FUNCTION_BLOCK FB_PcShutdownController
VAR
//---FB_Initで受け取り---
	_pPersistentDataManager		:POINTER TO FB_PersistentDataManager;		//パーシステントデータ書き込み
	_PcAmsNetId					:AMSNETID;									//PC AMS Net ID	

//---内部使用FB---
	fbPlcStop					:PLC_Stop		:=(Stop:=FALSE);			//PLCストップ
	fbNtShutdown				:NT_Shutdown	:=(START:=FALSE);			//PCシャットダウン
	fbNtReboot					:NT_Reboot		:=(START:=FALSE);			//PCリブート

	fbRebootTon					:TON			:=(PT:=T#2S);
	fbShutdownTon				:TON			:=(PT:=T#2S);
	
//---内部変数---
	iStep						:INT			:=0;						//シャットダウン、リブート制御step
	_bError						:BOOL;
	_bReboot					:BOOL;
	_bShutdown					:BOOL;
END_VAR

PROPERTY bError : BOOL
GET
bError:=_bError;
END_GET
END_PROPERTY

METHOD Execute
//---パーシステントデータ保存FBのポインターチェック---
	IF _pPersistentDataManager=0 THEN
		_bError:=TRUE;
		iStep:=0;
		RETURN;
		
	END_IF	



//---タイマーFB呼び出し---
	fbRebootTon(IN:=_bReboot AND NOT _bShutdown AND NOT _bError );
	fbShutdownTon(IN:=_bShutdown AND NOT _bReboot AND NOT _bError );



//---制御step---
	CASE iStep OF
		0:
			IF fbRebootTon.Q OR fbShutdownTon.Q THEN
				iStep:=10;
				
			END_IF
			
		10:				
			_pPersistentDataManager^.RequestWrite();
			iStep:=20;
	
		20:
			IF _pPersistentDataManager^.bWritePersistentDataDone THEN
				iStep:=30;
			ELSIF _pPersistentDataManager^.bWritePersistentDataError THEN
				_bError:=TRUE;
				iStep:=0;
			END_IF
		
		30:
		(*	fbPlcStop(	NETID	:=F_CreateAmsNetId(_PcAmsNetId),
						PORT	:=TwinCAT_SystemInfoVarList._AppInfo.AdsPort,
						Stop	:=_bReboot OR _bShutdown,
						TMOUT	:=DEFAULT_ADS_TIMEOUT,
						BUSY	=>,
						ERR		=>,
						ERRID	=>
						);
		*)
		
			fbNtReboot(	NETID	:=F_CreateAmsNetId(_PcAmsNetId),
						DELAY	:=1,
						START	:=_bReboot,
						TMOUT	:=DEFAULT_ADS_TIMEOUT,
						BUSY	=>,
						ERR		=>,
						ERRID	=>
						);
		
			fbNtShutdown(	NETID	:=F_CreateAmsNetId(_PcAmsNetId),
							DELAY	:=1,
							START	:=_bShutdown,
							TMOUT	:=DEFAULT_ADS_TIMEOUT,
							BUSY	=>,
							ERR		=>,
							ERRID	=>
							);
	
	END_CASE
END_METHOD

//FB_Init は常に暗黙的に使用可能で、主に初期化に使用されます。
//戻り値は評価されません。特定の結果を得るために、メソッドを明示的に宣言し、
//そのメソッドに標準の初期化コードをもったコードを追加することができます。戻り値を評価できます。
METHOD FB_Init: BOOL
VAR_INPUT
    bInitRetains: BOOL; // TRUE: 保持変数は初期化されます (ウォーム リセット、あるいはコールド リセット)
    bInCopyCode: BOOL;  // TRUE: 後でコードをコピーする (オンライン変更) ために、インスタンスをコピーします。

    pPersistentDataManager		:POINTER TO FB_PersistentDataManager;
	PcAmsNetId					:AMSNETID;		//PC AMS Net ID
END_VAR
_pPersistentDataManager := pPersistentDataManager;

_PcAmsNetId:=PcAmsNetId;
END_METHOD

METHOD  RequestReboot: BOOL
VAR_INPUT
	bExecute	:bool;
END_VAR
_bReboot		:=bExecute;
RequestReboot	:=bExecute;
END_METHOD

METHOD RequestShutdown: BOOL
VAR_INPUT
	bExecute	:BOOL;
END_VAR
_bShutdown			:=bExecute;
RequestShutdown		:=bExecute;
END_METHOD

METHOD ResetError
//エラー出力をリセット
_bError:=FALSE;
END_METHOD

END_FUNCTION_BLOCK

(* stored: Version 1.1.0.1
   POU FB_PcShutdownController: Id {5e504a49-c237-497e-bcc9-96deff8313f6}, SpecialFunc None
   Property bError: Id {2b3c858b-7971-4352-a5d1-6f1fe3c22d3c}
   Get Get: Id {505c4ddd-37bc-4ef5-9b1f-5b3a623797b9}
   Method Execute: Id {4fd55cde-97bb-4513-9a23-1b9ca06181b8}
   Method FB_Init: Id {4005cfe3-fa1e-4032-9be6-3c796e610e47}
   Method RequestReboot: Id {040fb411-3506-4400-b738-13ce029cde64}
   Method RequestShutdown: Id {c5c3a239-8c6b-4842-92ba-8cd5267593c6}
   Method ResetError: Id {e92edee7-e4c1-41c4-9428-960b4d095665} *)
